PROGRAM PRG_Simulator
VAR
	bInit					:BOOL := TRUE;					//Initialize

	fbItemGenerator			:FB_ItemGenerator;				//FB_ItemGenerator
	fbItemRegister			:FB_ItemRegister;				//FB_ItemRegister

	bStartGenerator			:BOOL;							// Start the generator
	bStopGenerator			:BOOL;							// Stop the generator

	bResetRegistry			:BOOL;							// Reset array registry

	stItemGen1 				: ST_ItemGenerator;				// Structure of generators
	stItemGen2 				: ST_ItemGenerator;
	stItemGen3 				: ST_ItemGenerator;
	stItemGen4 				: ST_ItemGenerator;
	stItemGen5 				: ST_ItemGenerator;
	stItemGen6 				: ST_ItemGenerator;
	stItemGen7 				: ST_ItemGenerator;
	stItemGen8 				: ST_ItemGenerator;
	stItemGen9 				: ST_ItemGenerator;
	stItemGen10 			: ST_ItemGenerator;
	stItemGenFromReg		: ST_ItemGenerator;
	
	aItemOnTimeRegistry		: ARRAY[0..GVL_Constant.ITEM_ARRAY_SIZE] OF TIME;		// Array of on time registrys
	aItemOffTimeRegistry	: ARRAY[0..GVL_Constant.ITEM_ARRAY_SIZE] OF TIME;		// Array of off time registrys
	nTimeCount				: INT;							// Count of total rising edge registrys
	osLoadOnTime			: F_TRIG;						// One shot load on time to generator
	osLoadOffTime			: R_TRIG;						// OIne shot load off time to generator
	i						: INT;							// Index container for array registrys
END_VAR

A_ItemGenerator();
A_ItemRegistry();

IF GVL_ItemSimulator.bResetRegistry AND NOT bResetRegistry THEN
	bResetRegistry := TRUE;
ELSE
	bResetRegistry := FALSE;
END_IF

ACTION A_ItemGenerator:
IF bInit THEN
	bInit := FALSE;
END_IF

//Number of pulses from registry
stItemGenFromReg.nNumberOfPulses := INT_TO_UINT(nTimeCount);

//One shots for loading on and off time
osLoadOnTime(CLK:=fbItemGenerator.bOutput);
osLoadOffTime(CLK:=fbItemGenerator.bOutput);

// Reset index
IF bResetRegistry OR i > nTimeCount OR bStartGenerator THEN
	i := 0;
	stItemGenFromReg.tTimeOnPulse := aItemOnTimeRegistry[i];
	stItemGenFromReg.tTimeOffPulse := aItemOffTimeRegistry[i+1];
END_IF;

//On bOutput falling edge
IF osLoadOnTime.Q AND stItemGenFromReg.bEnableGenerator THEN
	stItemGenFromReg.tTimeOnPulse := aItemOnTimeRegistry[i];
END_IF

// On bOutput rising edge
IF osLoadOffTime.Q AND stItemGenFromReg.bEnableGenerator THEN
	i := i + 1;
	stItemGenFromReg.tTimeOffPulse := aItemOffTimeRegistry[i];
END_IF





//Call Item generator program
fbItemGenerator(
	bStart:=bStartGenerator,
	bStop:=bStopGenerator,
	stItemGen1:=stItemGen1,
	stItemGen2:=stItemGen2,
	stItemGen3:=stItemGen3,
	stItemGen4:=stItemGen4,
	stItemGen5:=stItemGen5,
	stItemGen6:=stItemGen6,
	stItemGen7:=stItemGen7,
	stItemGen8:=stItemGen8,
	stItemGen9:=stItemGen9,
	stItemGen10:=stItemGen10,
	stItemGenFromReg:=stItemGenFromReg,
	bOutput=>GVL_ItemSimulator.bSignalOut);
	
	
//Reset start/stop
bStartGenerator := FALSE;
bStopGenerator := FALSE;
END_ACTION

ACTION A_ItemRegistry:
fbItemRegister(bSignal:=GVL_ItemSimulator.bSignalIn AND NOT fbItemGenerator.stItemGenFromReg.bEnableGenerator AND PRG_TCPIP.bConnectedCameraRead,
	bReset:=bResetRegistry,
	nTimeCount=>nTimeCount,
	aItemOnTimeRegistry=>aItemOnTimeRegistry,
	aItemOffTimeRegistry=>aItemOffTimeRegistry);
	
// Reset reset registry
bResetRegistry := FALSE;
END_ACTION

END_PROGRAM

(* stored: Version 1.1.0.1, ProductVersion 3.1.4024.12
   POU PRG_Simulator: Id {5a8209ee-df9d-4945-b39e-82e246e4b7c3}, SpecialFunc None
   Action A_ItemGenerator: Id {ea8d61fc-3f43-4c15-b430-7d59dc06e89a}
   Action A_ItemRegistry: Id {912b5aaf-f7c8-4236-8ccf-b7629f092d69} *)
